(*
:Description: function block for interpret the DPT from KNX devices
:Instructions for use: instantiate this function block to use the implemented interface I_KNX_DPT_Interpreter and its methods to interpret the KNX messages correctly
*)
FUNCTION_BLOCK KNX_DatapointTypes_Interpreter IMPLEMENTS I_KNX_DPT_Interpreter

METHOD M_InterpretAs2Bit : ST_KNX_DPT_B2
VAR_IN_OUT
	stInData		: ARRAY[*] OF BYTE;
END_VAR
M_InterpretAs2Bit.bBit1 := stInData[LOWER_BOUND(stInData,1)].0;
M_InterpretAs2Bit.bBit2 := stInData[LOWER_BOUND(stInData,1)].1;
END_METHOD

METHOD M_InterpretAsBool : BOOL
VAR_IN_OUT
	stInData		: ARRAY[*] OF BYTE;
END_VAR
M_InterpretAsBool := BYTE_TO_BOOL(stInData[LOWER_BOUND(stInData,1)]);
END_METHOD

METHOD M_InterpretAsDimming : ST_KNX_DPT_ControlDimming
VAR_IN_OUT
	stInData		: ARRAY[*] OF BYTE;
END_VAR
M_InterpretAsDimming.bControl 	:= stInData[LOWER_BOUND(stInData,1)].3;
M_InterpretAsDimming.nStepCode	:= stInData[LOWER_BOUND(stInData,1)] AND 16#07;
END_METHOD

METHOD M_InterpretAsFloat16 : REAL
VAR_IN_OUT
	stInData		: ARRAY[*] OF BYTE;
END_VAR
VAR
	nMantissa		: WORD;
	nSignMantissa	: INT;
	nExponent		: INT;
	fFloat			: REAL;
	nSign			: INT;
END_VAR
nSign 			:= BIT_TO_INT(stInData[LOWER_BOUND(stInData,1)].7);
nMantissa 		:= SHL(BYTE_TO_WORD(stInData[LOWER_BOUND(stInData,1)]) AND 16#07, 8);
nMantissa 		:= nMantissa OR BYTE_TO_WORD(stInData[LOWER_BOUND(stInData,1) + 1]);
nSignMantissa 	:= WORD_TO_INT(nMantissa);
IF nSign = 1 THEN
	// negative value
	nMantissa := NOT nMantissa;
	nMantissa := nMantissa OR (NOT 16#F800);
	nSignMantissa := WORD_TO_INT(nMantissa + 1);
	nSignMantissa := nSignMantissa * -1;
END_IF
nExponent := BYTE_TO_INT(stInData[LOWER_BOUND(stInData,1)] AND 16#78);
M_InterpretAsFloat16 := LREAL_TO_REAL(0.01 * nSignMantissa * EXPT(2, nExponent));
END_METHOD

METHOD M_InterpretAsINT16 : INT
VAR_IN_OUT
	stInData		: ARRAY[*] OF BYTE;
END_VAR
VAR
	nResult			: WORD;
END_VAR
nResult := SHL(BYTE_TO_WORD(stInData[LOWER_BOUND(stInData,1)]), 8);
nResult := nResult OR BYTE_TO_WORD(stInData[LOWER_BOUND(stInData,1)+1]);
M_InterpretAsINT16 := WORD_TO_INT(nResult);
END_METHOD

METHOD M_InterpretAsINT32 : DINT
VAR_IN_OUT
	stInData		: ARRAY[*] OF BYTE;
END_VAR
VAR
	nResult			: DWORD;
END_VAR
nResult := SHL(BYTE_TO_DWORD(stInData[LOWER_BOUND(stInData,1)]), 8*3);
nResult := nResult OR SHL(BYTE_TO_DWORD(stInData[LOWER_BOUND(stInData,1)+1]), 8*2);
nResult := nResult OR SHL(BYTE_TO_DWORD(stInData[LOWER_BOUND(stInData,1)+2]), 8);
nResult := nResult OR BYTE_TO_DWORD(stInData[LOWER_BOUND(stInData,1)+3]);
M_InterpretAsINT32 := DWORD_TO_DINT(nResult);
END_METHOD

METHOD M_InterpretAsUINT16 : UINT
VAR_IN_OUT
	stInData		: ARRAY[*] OF BYTE;
END_VAR
VAR
	nResult			: UINT;
END_VAR
nResult := SHL(BYTE_TO_WORD(stInData[LOWER_BOUND(stInData,1)]),8);
nResult := nResult OR BYTE_TO_WORD(stInData[LOWER_BOUND(stInData,1)+1]);
M_InterpretAsUINT16 := nResult;
END_METHOD

METHOD M_InterpretAsUINT32 : UDINT
VAR_IN_OUT
	stInData		: ARRAY[*] OF BYTE;
END_VAR
VAR
	nResult			: UDINT;
END_VAR
nResult := SHL(BYTE_TO_DWORD(stInData[LOWER_BOUND(stInData,1)]),8*3);
nResult := nResult OR SHL(BYTE_TO_DWORD(stInData[LOWER_BOUND(stInData,1)]+1),8*2);
nResult := nResult OR SHL(BYTE_TO_DWORD(stInData[LOWER_BOUND(stInData,1)]+2),8);
nResult := nResult OR BYTE_TO_DWORD(stInData[LOWER_BOUND(stInData,1)]+3);
M_InterpretAsUINT32 := nResult;
END_METHOD

METHOD M_InterpretAsUINT8 : BYTE
VAR_IN_OUT
	stInData		: ARRAY[*] OF BYTE;
END_VAR
M_InterpretAsUINT8 := stInData[LOWER_BOUND(stInData,1)];
END_METHOD

METHOD M_InterpretNewMessage : BOOL
VAR_INPUT
	stInData		: BOOL;
END_VAR
M_InterpretNewMessage := stInData;
END_METHOD

END_FUNCTION_BLOCK

(* stored: Version 1.1.0.1
   POU KNX_DatapointTypes_Interpreter: Id {64a4add0-5fc0-47d2-9b2b-aa98e64f4a8b}, SpecialFunc None
   Method M_InterpretAs2Bit: Id {645492f9-18c4-4f90-8fb1-b54d58cb0e2d}
   Method M_InterpretAsBool: Id {2ddcc710-928d-48c3-a3f6-c43b38918035}
   Method M_InterpretAsDimming: Id {143d9181-0d00-4d88-a1c7-34f12b72adf9}
   Method M_InterpretAsFloat16: Id {53d6f035-7a63-4f7b-854c-2433a97caaa2}
   Method M_InterpretAsINT16: Id {0b31627f-6e0f-441c-bfc7-ded814e29f56}
   Method M_InterpretAsINT32: Id {807cc6c2-55d5-47f3-b81a-90819bbd727c}
   Method M_InterpretAsUINT16: Id {c5321905-d1cb-401c-8b44-6c7dd303848c}
   Method M_InterpretAsUINT32: Id {766d3e75-e0c8-4fec-af38-156e514382ed}
   Method M_InterpretAsUINT8: Id {96608cde-e332-45f2-af3d-3230e4e9dcea}
   Method M_InterpretNewMessage: Id {0e3df83d-fa35-48fa-b003-a58eab4d369e} *)
